// Mitsubishi GX Works2 project: b01   PLC: Q02/Q02H

PROGRAM MAIN
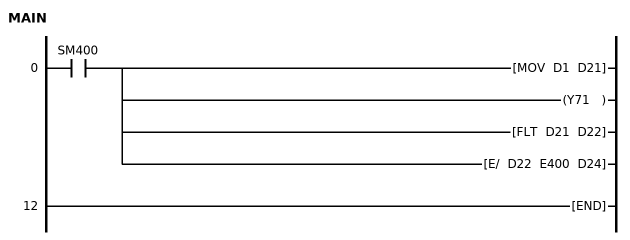
0     LD      SM400
      MOV     D1 D21
      OUT     Y71
      FLT     D21 D22
      E/      D22 E400 D24
12    END
END_PROGRAM
